(* Logix 5000 project; controller START_STOP Emulate 5570 rev 30.12; software revision 30.00 *)

TASK MainTask (continuous, watchdog 500 ms) : MainProgram

MODULES
   Local : Emulate 5570 (ICP 2, rev 30.12)
      VIRTUAL_OUTPUTS : vendor 1 type 0 code 15 (ICP 4, rev 1.1, Output RPI 50 ms)
      VIRTUAL_INPUTS : vendor 1 type 0 code 15 (ICP 3, rev 1.1, Output RPI 50 ms)
END_MODULES

VAR_GLOBAL   (* controller tags *)
   CCR : BOOL;
   CVY_1 : ALIAS FOR Local:4:O.Data[0].7;
   CVY_1_2_DN : BOOL;
   CVY_2 : ALIAS FOR Local:4:O.Data[0].8;
   CVY_20 : ALIAS FOR Local:4:O.Data[0].4;
   CVY_21 : ALIAS FOR Local:4:O.Data[0].5;
   CVY_22 : ALIAS FOR Local:4:O.Data[0].6;
   CVY_22_DN : BOOL;
   CVY_3 : ALIAS FOR Local:4:O.Data[0].9;
   CVY_3_DN : BOOL;
   CVY_4 : ALIAS FOR Local:4:O.Data[0].10;
   CVY_4_DN : BOOL;
   CVY_5 : ALIAS FOR Local:4:O.Data[0].11;
   CVY_5_DN : BOOL;
   CVY_8 : ALIAS FOR Local:4:O.Data[0].3;
   CVY_8_DN : BOOL;
   DEL_1 : TIMER := (PRE := 1000);
   DEL_2 : TIMER := (PRE := 1000);
   DEL_3 : TIMER := (PRE := 1000);
   DEL_4 : TIMER := (PRE := 1000);
   DEL_5 : TIMER := (PRE := 1000);
   DEL_7 : TIMER := (PRE := 1000);
   FIN_SP1 : ALIAS FOR Local:3:I.Data[1].2;
   FIN_SP2 : ALIAS FOR Local:3:I.Data[1].3;
   PB_CVY_1 : ALIAS FOR Local:3:I.Data[1].8;
   PB_CVY_2 : ALIAS FOR Local:3:I.Data[1].9;
   PB_CVY_22 : ALIAS FOR Local:3:I.Data[1].5;
   PB_CVY_3 : ALIAS FOR Local:3:I.Data[1].12;
   PB_CVY_4 : ALIAS FOR Local:3:I.Data[1].14;
   PB_CVY_5 : ALIAS FOR Local:3:I.Data[1].16;
   PB_CVY_8 : ALIAS FOR Local:3:I.Data[1].4;
   PRUEBA : BOOL;
   SNR_CVY_1 : ALIAS FOR Local:3:I.Data[1].10;
   SNR_CVY_2 : ALIAS FOR Local:3:I.Data[1].11;
   SNR_CVY_22 : ALIAS FOR Local:3:I.Data[1].7;
   SNR_CVY_3 : ALIAS FOR Local:3:I.Data[1].13;
   SNR_CVY_4 : ALIAS FOR Local:3:I.Data[1].15;
   SNR_CVY_5 : ALIAS FOR Local:3:I.Data[1].17;
   SNR_CVY_8 : ALIAS FOR Local:3:I.Data[1].6;
   SP1_DN : BOOL;
   SP2_DN : BOOL;
   SR1 : BOOL;
   SR13 : BOOL;
   SR18 : BOOL;
   SR19 : BOOL;
   SR2 : BOOL;
   SR3 : BOOL;
   SR33 : BOOL;
   SR4 : BOOL;
   SR5 : BOOL;
   SR6 : BOOL;
   Started : ALIAS FOR Local:4:O.Data[0].0;
   STP_g : ALIAS FOR Local:3:I.Data[1].1;
   STT_g : ALIAS FOR Local:3:I.Data[1].0;
   STT_SP1 : ALIAS FOR Local:4:O.Data[0].1;
   STT_SP2 : ALIAS FOR Local:4:O.Data[0].2;
   TF_1 : TIMER := (PRE := 2000);
   TF_2 : TIMER := (PRE := 2000);
   TF_3 : TIMER := (PRE := 2000);
   TRN_33_DN : BOOL;
   TRN_3_DN : BOOL;
   TRN_4_DN : BOOL;
END_VAR

PROGRAM MainProgram   (* main routine MainRoutine *)

ROUTINE Encendido_CVY22   (* ladder *)
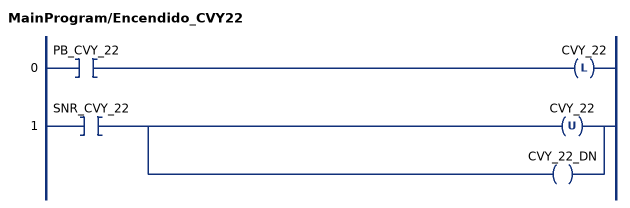
   0: XIC(PB_CVY_22)OTL(CVY_22);
   1: XIC(SNR_CVY_22)[OTU(CVY_22) ,OTE(CVY_22_DN) ];
END_ROUTINE

ROUTINE Encendido_CVY4   (* ladder *)
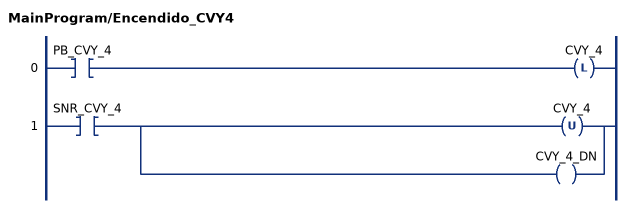
   0: XIC(PB_CVY_4)OTL(CVY_4);
   1: XIC(SNR_CVY_4)[OTU(CVY_4) ,OTE(CVY_4_DN) ];
END_ROUTINE

ROUTINE Encendido_CVY5   (* ladder *)
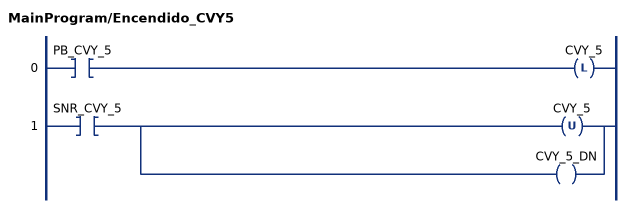
   0: XIC(PB_CVY_5)OTL(CVY_5);
   1: XIC(SNR_CVY_5)[OTU(CVY_5) ,OTE(CVY_5_DN) ];
END_ROUTINE

ROUTINE Encendido_CVY8   (* ladder *)
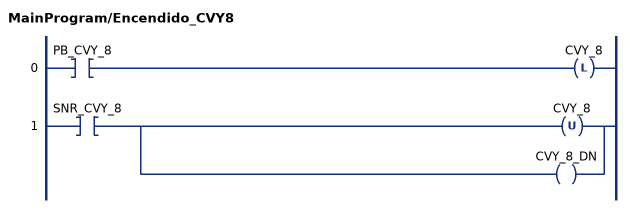
   0: XIC(PB_CVY_8)OTL(CVY_8);
   1: XIC(SNR_CVY_8)[OTU(CVY_8) ,OTE(CVY_8_DN) ];
END_ROUTINE

ROUTINE Inicio_Soplado   (* ladder *)
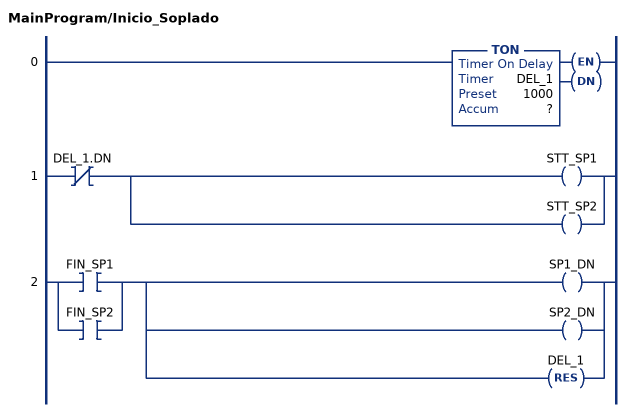
   0: TON(DEL_1,?,?);
   1: XIO(DEL_1.DN)[OTE(STT_SP1) ,OTE(STT_SP2) ];
   2: [XIC(FIN_SP1) ,XIC(FIN_SP2) ][OTE(SP1_DN) ,OTE(SP2_DN) ,RES(DEL_1) ];
END_ROUTINE

ROUTINE MainRoutine   (* ladder *)
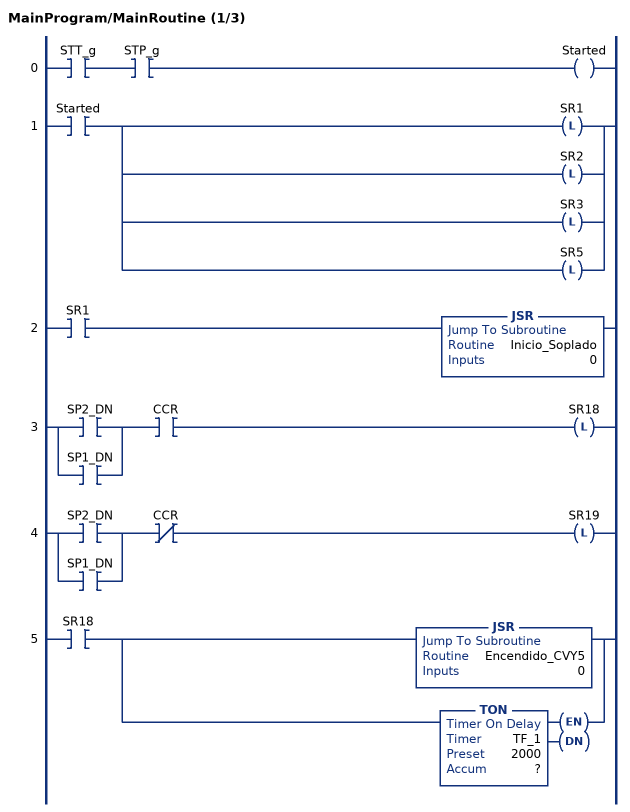
   0: XIC(STT_g)XIC(STP_g)OTE(Started);
   1: XIC(Started)[OTL(SR1) ,OTL(SR2) ,OTL(SR3) ,OTL(SR5) ];
   2: XIC(SR1)JSR(Inicio_Soplado,0);
   3: [XIC(SP2_DN) ,XIC(SP1_DN) ]XIC(CCR)OTL(SR18);
   4: [XIC(SP2_DN) ,XIC(SP1_DN) ]XIO(CCR)OTL(SR19);
   5: XIC(SR18)[JSR(Encendido_CVY5,0) ,TON(TF_1,?,?) ];
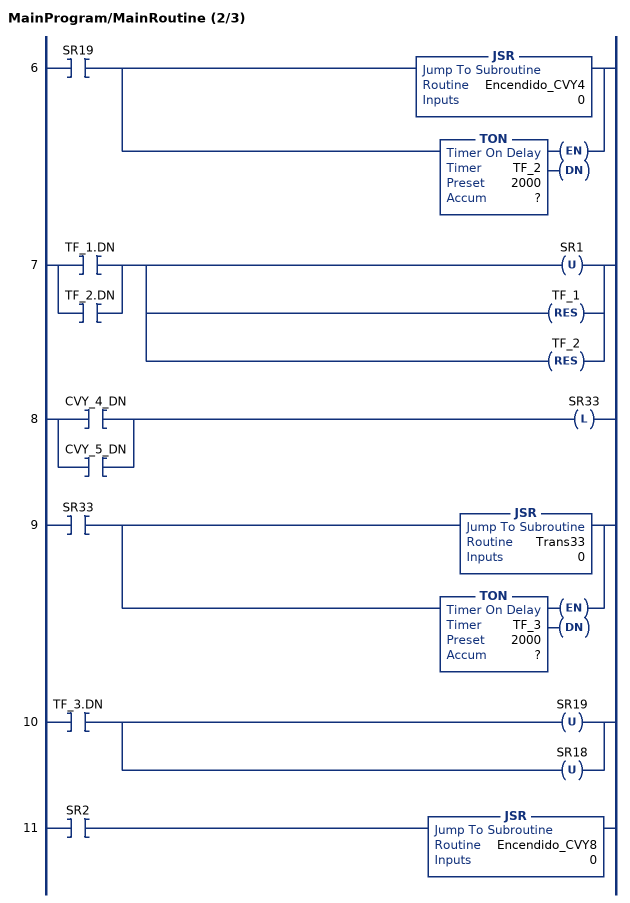
   6: XIC(SR19)[JSR(Encendido_CVY4,0) ,TON(TF_2,?,?) ];
   7: [XIC(TF_1.DN) ,XIC(TF_2.DN) ][OTU(SR1) ,RES(TF_1) ,RES(TF_2) ];
   8: [XIC(CVY_4_DN) ,XIC(CVY_5_DN) ]OTL(SR33);
   9: XIC(SR33)[JSR(Trans33,0) ,TON(TF_3,?,?) ];
   10: XIC(TF_3.DN)[OTU(SR19) ,OTU(SR18) ];
   11: XIC(SR2)JSR(Encendido_CVY8,0);
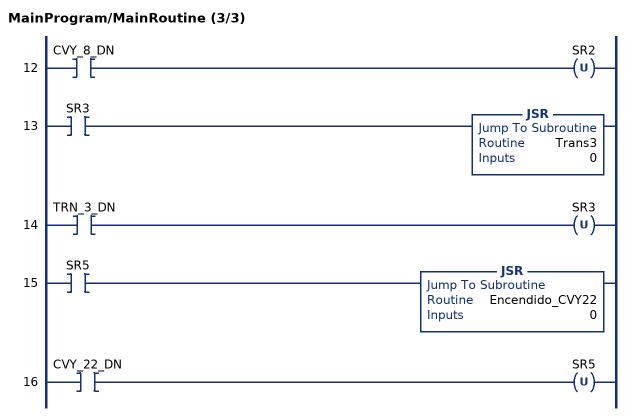
   12: XIC(CVY_8_DN)OTU(SR2);
   13: XIC(SR3)JSR(Trans3,0);
   14: XIC(TRN_3_DN)OTU(SR3);
   15: XIC(SR5)JSR(Encendido_CVY22,0);
   16: XIC(CVY_22_DN)OTU(SR5);
END_ROUTINE

ROUTINE Trans3   (* ladder *)
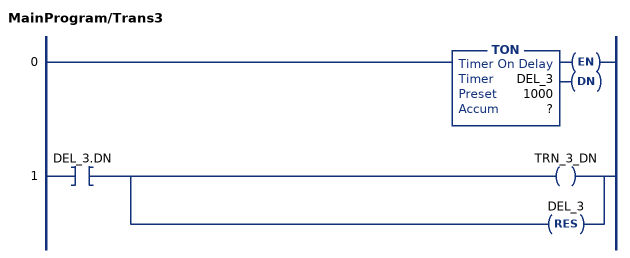
   0: TON(DEL_3,?,?);
   1: XIC(DEL_3.DN)[OTE(TRN_3_DN) ,RES(DEL_3) ];
END_ROUTINE

ROUTINE Trans33   (* ladder *)
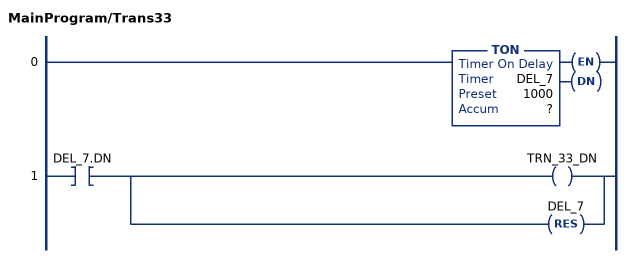
   0: TON(DEL_7,?,?);
   1: XIC(DEL_7.DN)[OTE(TRN_33_DN) ,RES(DEL_7) ];
END_ROUTINE
END_PROGRAM
